(* PLC project CoDeSys External Library Template, WAGO e!COCKPIT e!COCKPIT, author 3S - Smart Software Solutions GmbH *)
(* stored: creationDateTime 2019-10-29T12:22:40.9919411, version 3.5.5.30, modificationDateTime 2019-10-24T14:40:07.960949, organization 3S - Smart Software Solutions GmbH *)
(* Library project template with all possible element types, docu and a sample project structure *)

FUNCTION fnZlozenieBitowWRejestr16Bit : BOOL
  VAR_INPUT
    xBit0 : BOOL;
    xBit1 : BOOL;
    xBit2 : BOOL;
    xBit3 : BOOL;
    xBit4 : BOOL;
    xBit5 : BOOL;
    xBit6 : BOOL;
    xBit7 : BOOL;
    xBit8 : BOOL;
    xBit9 : BOOL;
    xBit10 : BOOL;
    xBit11 : BOOL;
    xBit12 : BOOL;
    xBit13 : BOOL;
    xBit14 : BOOL;
    xBit15 : BOOL;
  END_VAR
  VAR_OUTPUT
    wRejestr16Bit : WORD;
  END_VAR

            (*			
Autor:					Paweł Kąkol, 
Prawa majątkowe: 		Solwena Sp. z o.o., 
Aktualizacje:			2017-12-13-09:30-PK - stworzenie

Opis:					Funkcja do składania rejestru 16-bitowego typu WORD z pojedynczych zmiennych BOOL,
						Nalezy pamietac, ze numeracja bitow jest zgodna z odpowiadajacymi wykladnikami potegi liczby 2
*)
wRejestr16Bit := 0;
//sprawdzanie stanu bitow
IF xBit0 THEN
	wRejestr16Bit := 1;	
END_IF
IF xBit1 THEN
	wRejestr16Bit := wRejestr16Bit + 2;	
END_IF
IF xBit1 THEN
	wRejestr16Bit := wRejestr16Bit + 4;	
END_IF
IF xBit1 THEN
	wRejestr16Bit := wRejestr16Bit + 8;	
END_IF
IF xBit1 THEN
	wRejestr16Bit := wRejestr16Bit + 16;	
END_IF
IF xBit1 THEN
	wRejestr16Bit := wRejestr16Bit + 32;	
END_IF
IF xBit1 THEN
	wRejestr16Bit := wRejestr16Bit + 64;	
END_IF
IF xBit1 THEN
	wRejestr16Bit := wRejestr16Bit + 128;	
END_IF
IF xBit1 THEN
	wRejestr16Bit := wRejestr16Bit + 256;	
END_IF
IF xBit1 THEN
	wRejestr16Bit := wRejestr16Bit + 512;	
END_IF
IF xBit1 THEN
	wRejestr16Bit := wRejestr16Bit + 1024;	
END_IF
IF xBit1 THEN
	wRejestr16Bit := wRejestr16Bit + 2048;	
END_IF
IF xBit1 THEN
	wRejestr16Bit := wRejestr16Bit + 4096;	
END_IF
IF xBit1 THEN
	wRejestr16Bit := wRejestr16Bit + 8192;	
END_IF
IF xBit1 THEN
	wRejestr16Bit := wRejestr16Bit + 16384;	
END_IF
IF xBit1 THEN
	wRejestr16Bit := wRejestr16Bit + 32768;	
END_IF
          
END_FUNCTION
